Staubli VAL3: numericalTwins.pjx

--- numericalTwins.pjx ---
Parameters version=s7.11.3 stackSize=5000 millimeterUnit=true
Program file=init.pgx
Program file=start.pgx
Program file=stop.pgx
Program file=tPosition.pgx
Program file=tRobot.pgx
Data file=numericalTwins.dtx

--- numericalTwins.dtx ---
mdesc mNomSpeed
sio sioSocket = {link=Socket\test}
jointRx jHere
string sData
num nFrameIndex
num nEol
string sTaskPos
bool bOvrPosition
num nOvrPos
num nPrevOvrPos
string sTaskRobot
jointRx jStart
pointRx pPick = {fatherId=world[0]}
trsf trAppro
pointRx pPlace = {fatherId=world[0]}

--- start.pgx ---
program start()
begin
  // Initialisation
  call init()

  // Creation tache suivi position toutes les 4ms
  taskCreateSync sTaskPos, 0.004, bOvrPosition, tPosition()

  // On attend qu'elle soit démarree
  wait(taskStatus(sTaskPos)==1)



  // Lancement du process principal
  taskCreate sTaskRobot, 100, tRobot()
  wait(taskStatus(sTaskRobot)==1)

  // Surveillance
  while true
    if nPrevOvrPos!=nOvrPos
      logMsg("Overrun dans la tache "+sTaskPos)
      nPrevOvrPos=nOvrPos
    endIf

    delay(0)
  endWhile
end

--- init.pgx ---
program init()
begin
  // Initialise toutes les variables

  // Nom des taches
  sTaskPos="tPosition"
  sTaskRobot="tRobot"
  // Booleen de detection overrun de la tache
  bOvrPosition=false
  // Suivi des overrun par l'application
  nOvrPos=0
  nPrevOvrPos=0
  // Numero de la trame
  nFrameIndex=0
  // Caractere de fin de chaine LF, code 10 en decimal
  nEol=10
  // Pour la communication socket
  // La baie est client TCP, elle discute avec le serveur TCP
  // a l'adresse IP "on met l'adresse ip du pc qui fera serveur", sur le port 2005
  // On fait une ecriture en continu, pas de timeout
  sioCtrl(sioSocket,"port",2005)
  sioCtrl(sioSocket,"target","192.168.0.3")
  sioCtrl(sioSocket,"endOfString",nEol)
  sioCtrl(sioSocket,"timeout",-1)
  sioCtrl(sioSocket,"nagle",false)

  // trsf d'approche
  trAppro={0,0,-50,0,0,0}
end

--- tPosition.pgx ---
program tPosition()
  local num l_nIndex
begin
  // La trame envoye au serveur aura la structure:
  // {index;j1;j2;j3;j4;j5;j6}
  // { = debut de chaine
  // } = fin de chaine
  // ; separateur de donnees
  // index = numero de la trame pour voir si perte
  // j1, j2, j3, j4, j5, j6: position de chaque joint

  while true
    delay(0)

    nFrameIndex = nFrameIndex + 1

    // On recupere la position robot en joint
    jHere=herej()

    // On recupere la position robot en cartésien (x,y,z,Rx,Ry,Rz)
    pHere = here(torche, world)



    // On construit la chaine /!\ 128 caractere maxi
    sData="{"
    sData=sData+toString("",nFrameIndex)+";"
    sData=sData+toString("10.3",jHere.j1)+";"
    sData=sData+toString("10.3",jHere.j2)+";"
    sData=sData+toString("10.3",jHere.j3)+";"
    sData=sData+toString("10.3",jHere.j4)+";"
    sData=sData+toString("10.3",jHere.j5)+";"
    sData=sData+toString("10.3",jHere.j6)+"}"

    // Coordonnées Cartésiennes (X, Y, Z, RX, RY, RZ)
    sData = sData + toString(".3", pHere.trsf.x) + ";"
    sData = sData + toString(".3", pHere.trsf.y) + ";"
    sData = sData + toString(".3", pHere.trsf.z) + ";"
    sData = sData + toString(".3", pHere.trsf.rx) + ";"
    sData = sData + toString(".3", pHere.trsf.ry) + ";"
    sData = sData + toString(".3", pHere.trsf.rz) + "}"

    // On envoie la trame
    for l_nIndex=0 to len(sData)-1
      sioSet(sioSocket,asc(sData,l_nIndex))
    endFor
    // On envoie une fin de chaine
    sioSet(sioSocket,nEol)

    // Si depassement de temps, on incremente
    if bOvrPosition
      nOvrPos=nOvrPos+1
    endIf
  endWhile
end

--- tRobot.pgx ---
program tRobot()
begin
  resetMotion(jStart)

  while true
    movej(appro(pPick,trAppro),flange,mNomSpeed)
    movel(pPick,flange,mNomSpeed)
    waitEndMove()
    movel(appro(pPick,trAppro),flange,mNomSpeed)

    movej(appro(pPlace,trAppro),flange,mNomSpeed)
    movel(pPlace,flange,mNomSpeed)
    waitEndMove()
    movel(appro(pPlace,trAppro),flange,mNomSpeed)

    delay(0)
  endWhile
end
